(* IEC 61131-3 sources: pub-control-lib/src/Interfaces/PubControl, 2 files *)

(* ---- ITank.st ---- *)
USING Siemens.PubControl.Types;
USING Siemens.PubControl.Types;

NAMESPACE Siemens.PubControl.Interfaces

    INTERFACE ITank
        METHOD SetMaxLevel : INT
            VAR_INPUT
                MaxLevel : UINT;
            END_VAR
        END_METHOD

        METHOD GetLevel : UINT
        END_METHOD

        METHOD GetStatus : TankStatus
        END_METHOD

        METHOD Cleaning
            VAR_INPUT
                Start : BOOL;
                Stop : BOOL;
            END_VAR
        END_METHOD

        METHOD Tanking
        END_METHOD
    END_INTERFACE

END_NAMESPACE

(* ---- ITapBar.st ---- *)
NAMESPACE Siemens.PubControl.Interfaces
    INTERFACE ITapBar

        METHOD CalcImpulses
            VAR_INPUT
                MeasureTime : LTIME;
                Impulses : INT;
                Factor : INT;
            END_VAR

        END_METHOD

        METHOD GetConsumption : Real
        END_METHOD

        METHOD GetFlow : Real
        END_METHOD

        METHOD Reset
        END_METHOD

    END_INTERFACE

END_NAMESPACE
